ADAPTER IGritScreenFlushing (* Adapter Interface *)
  (* Standard: 61499-1 *)
  (* Version 0.0, 7/6/2026, Schneider Electric *)
  PACKAGE SE.Nereda;
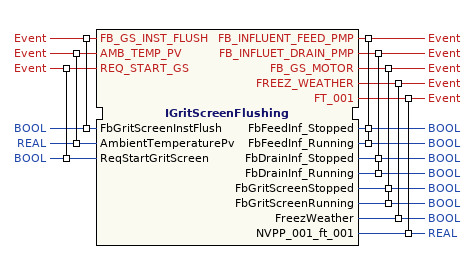
  EVENT_INPUT
    FB_GS_INST_FLUSH WITH FbGritScreenInstFlush;
    AMB_TEMP_PV WITH AmbientTemperaturePv;
    REQ_START_GS WITH ReqStartGritScreen;
  END_EVENT
  EVENT_OUTPUT
    FB_INFLUENT_FEED_PMP WITH FbFeedInf_Stopped, FbFeedInf_Running;
    FB_INFLUET_DRAIN_PMP WITH FbDrainInf_Stopped, FbDrainInf_Running;
    FB_GS_MOTOR WITH FbGritScreenStopped, FbGritScreenRunning;
    FREEZ_WEATHER WITH FreezWeather;
    FT_001 WITH NVPP_001_ft_001;
  END_EVENT
  VAR_INPUT
    FbGritScreenInstFlush : BOOL;
    AmbientTemperaturePv : REAL;
    ReqStartGritScreen : BOOL;
  END_VAR
  VAR_OUTPUT
    FbFeedInf_Stopped : BOOL;
    FbFeedInf_Running : BOOL;
    FbDrainInf_Stopped : BOOL;
    FbDrainInf_Running : BOOL;
    FbGritScreenStopped : BOOL;
    FbGritScreenRunning : BOOL;
    FreezWeather : BOOL;
    NVPP_001_ft_001 : REAL;
  END_VAR
  SERVICE SOCKET/PLUG
    SEQUENCE request_confirm
      SOCKET.REQ(REQD) -> PLUG.REQ(REQD);
      PLUG.CNF(CNFD) -> SOCKET.CNF(CNFD);
    END_SEQUENCE
    SEQUENCE indication_response
      PLUG.IND(INDD) -> SOCKET.IND(INDD);
      SOCKET.RSP(RSPD) -> PLUG.RSP(RSPD);
    END_SEQUENCE
  END_SERVICE
END_ADAPTER
